// TIA Portal project "FuncionesTIAPortal" (V17)

(* hardware
DEVICE "S7-1500/ET200MP station_1"  S7-1500 station
   slot 0: "Rail_0"  Rack  6ES7 590-1***0-0AA0
   slot 1: "PLC_1"  CPU 1515-2 PN  6ES7 515-2AM00-0AB0  V1.8
      slot 3: "CPU display_1"  6ES7591-1BA00-0AA0
      slot 32768: "PROFINET interface_1"  X1
         slot 32769: "Port_1"  X1 P1
         slot 32770: "Port_2"  X1 P2
      slot 33024: "PROFINET interface_2"  X2
         slot 33025: "Port_1"  X2 P1
*)

// ===== PLC "PLC_1"  CPU 1515-2 PN =====

VAR_GLOBAL   // PLC tag table "Default tag table"
   "arranque" AT %E0.0 : Bool;
   "Tag_2" AT %E0.1 : Bool;
   "motor1" AT %A0.0 : Bool;
   "Tag_4" AT %M0.0 : Bool;
   "Tag_5" AT %Z1 : Counter;
   "Tag_6" AT %T1 : Timer;
   "Tag_7" AT %E0.2 : Bool;
   "ciclo1" AT %E1.0 : Bool;
   "ciclo2" AT %E1.1 : Bool;
   "Tag_10" AT %T2 : Timer;
   "Tag_11" AT %T3 : Timer;
   "motor2" AT %A0.1 : Bool;
   "motor3" AT %A0.2 : Bool;
   "start" AT %E0.3 : Bool;
END_VAR

FUNCTION "funcionamientoMotores" : Void   // FC1, STL
TITLE = LOGICA DE MOTORES CON TIEMPOS
{ S7_Optimized_Access := 'TRUE' }
AUTHOR : Luis Hernandez
VERSION : 0.1
// TRES MOTORES CON DIFERENTES TIEMPOS SECUENCIADOS
   VAR_INPUT
      tmotor1 : S5Time;
      tmotor2 : S5Time;
      tmotor3 : S5Time;
   END_VAR
BEGIN

REGION Network 1
         A     "start";  //arranque

         L     #tmotor1;
         SP    "Tag_6";

         L     #tmotor2;
         SP    "Tag_10";

         L     #tmotor3;
         SP    "Tag_11";

         A     "Tag_6";
         =     "motor1";

         A     "Tag_10";
         =     "motor2";

         A     "Tag_11";
         =     "motor3";
END_REGION
END_FUNCTION

ORGANIZATION_BLOCK "Main"   // OB1, LAD, ProgramCycle
TITLE = "Main Program Sweep (Cycle)"
{ S7_Optimized_Access := 'TRUE' }
VERSION : 0.1
   VAR_INPUT
      Initial_Call : Bool;   // Initial call of this OB
      Remanence : Bool;   // =True, if remanent data are available
   END_VAR
BEGIN

REGION Network 2 (STL)
         A     "Tag_2";
         CU    "Tag_5";

         A     "Tag_7";
         CD    "Tag_5";

         L     1;
         L     "Tag_5";
         ==I;
         A     "start";
         JC    motor1;

         L     2;
         L     "Tag_5";
         ==I;
         A     "start";
         JC    motor2;

         L     3;
         L     "Tag_5";
         ==I;
         A     "start";
         JC    motor3;



   motor1:CALL  "funcionamientoMotores"
         ( tmotor1 := S5T#5s,
           tmotor2 := S5T#8s,
           tmotor3 := S5T#20s
         );

   motor2:CALL  "funcionamientoMotores"
         ( tmotor1 := S5T#7s,
           tmotor2 := S5T#6s,
           tmotor3 := S5T#8s
         );

   motor3:CALL  "funcionamientoMotores"
         ( tmotor1 := S5T#4s,
           tmotor2 := S5T#12s,
           tmotor3 := S5T#15s
         );
END_REGION
END_ORGANIZATION_BLOCK